(* IEC 61131-3 sources: Industry-PLC-LLM/data/PLCBEAD_repo/PLCBEAD_PLCEmbed-main/PLC-BEAD/Source/GEB/TRUNC_REAL, 1 file *)

(* ---- TRUNC_REAL.ST ---- *)
FUNCTION TRUNC_REAL:REAL

	VAR_INPUT
		IN :	REAL;
	END_VAR

	TRUNC_REAL := UDINT_TO_REAL(DINT_TO_UDINT(TRUNC(IN)));
END_FUNCTION

PROGRAM program0

	VAR
		IN :	REAL;
		OUT: REAL;
	END_VAR
	OUT := TRUNC_REAL(IN);

END_PROGRAM
